{attribute 'qualified_only'}
TYPE E_LogType:
(
	Info := 1, 
	Warnung := 2, 
	Fehler := 3
) BYTE;
END_TYPE

(* stored: Version 1.1.0.1, ProductVersion 3.1.4024.2
   DUT E_LogType: Id {89b7e1f1-2019-47ac-9aa6-96579890ea36} *)
